{attribute 'qualified_only'}
{attribute 'strict'}
{attribute 'to_string'}
TYPE E_SeqAX5000 :
(
	{warning '#TODO: update during development'}
	INIT := 0,
	STOPPED,
	BUSY,
	STOPPING,
	ERROR
);
END_TYPE

(* stored: Version 1.1.0.1, ProductVersion 3.1.4024.12
   DUT E_SeqAX5000: Id {c09962e6-f12f-412b-870f-0456e90e688d} *)
